# EPICS substitutions: iocs/MC06/db/SAI_DigitalChannels.substitutions
file /opt/epics/modules/SAI/db/SAI_DigitalChannels.template {
pattern {	P,		R,		SCAN, 		ASYNPORT}
        { 	"XF:06BM-BI",		"{MC:06}",	"1 second",	"pmac"}
}

#EOF
